FUNCTION_BLOCK PressureSensor IMPLEMENTS ITF_AnalogSensor
VAR_INPUT
END_VAR
VAR_OUTPUT
END_VAR
VAR
	//Hardware
	AI_CurrentPressure AT %I* : INT;
END_VAR

PROPERTY Value : INT
GET
Value := AI_CurrentPressure;
END_GET
END_PROPERTY

END_FUNCTION_BLOCK

(* stored: Version 1.1.0.1, ProductVersion 3.1.4024.9
   POU PressureSensor: Id {0cf60463-ace6-4c96-91c5-54c6f310aeb6}, SpecialFunc None
   Property Value: Id {1ec48ceb-72ca-434b-9146-7f6a915f7385}
   Get Get: Id {2524344c-0044-4014-ad0f-9ea03ea63af5} *)
